PROGRAM P_Demo_UInt64Limit
VAR
    uliRpmMin   : T_ULARGE_INTEGER;; // 转速下限 100
    uliRpmMax   : T_ULARGE_INTEGER;; // 转速上限 5000
    uliHmiInput : T_ULARGE_INTEGER;; // 操作员输入
    uliRpmSafe  : T_ULARGE_INTEGER;; // 限幅后
    bLimit      : BOOL;
END_VAR

// ============================================================
// Tc2_Utilities.UInt64Limit 演示程序（FUNCTION，单周期触发）
// ============================================================
// 场景：HMI 操作员输入电机转速设定值，必须裁剪到机械允许的最大转速 5000 rpm = 5000，最小 100。
// 价值：替代手写两次 `UInt64Cmp64` + 嵌套 IF；一次调用语义清晰。
// 验证步骤：
//   1. 把本 PROGRAM 加到 PlcTask 调用列表
//   2. 编译 + 登录
//   3. 在线把 b... 触发位置 TRUE 一个周期
//   4. 观察输出变量是否符合期望
// ============================================================

uliRpmMin := ULARGE_INTEGER(0, 100);
uliRpmMax := ULARGE_INTEGER(0, 5000);
IF bLimit THEN
    // 防止操作员误输入超界值打坏机械
    uliRpmSafe := UInt64Limit(uliRpmMin, uliHmiInput, uliRpmMax);
    bLimit := FALSE;
END_IF;

END_PROGRAM

(* stored: Version 1.1.0.1, ProductVersion 3.1.4024.5
   POU P_Demo_UInt64Limit: Id {fe75f5d4-82d0-55cd-af7e-6cb601a6e7ae}, SpecialFunc None *)
